                               // Now build the request data
                               #V_PN_Measurement_Data_2.Service_Data_Request.Count_Meas_Values := INT_TO_BYTE(#RECORD_PE_COUNT_MEAS_2);
                               #V_PN_Measurement_Data_2.Service_Data_Request.Meas_Values[PE_ID_F_MAX] := 61;
                               #V_PN_Measurement_Data_2.Service_Data_Request.Meas_Values[PE_ID_U_AVG_L_N_MAX] := 62;
                               #V_PN_Measurement_Data_2.Service_Data_Request.Meas_Values[PE_ID_U_AVG_L_L_MAX] := 63;
                               #V_PN_Measurement_Data_2.Service_Data_Request.Meas_Values[PE_ID_I_AVG_MAX] := 64;
                               #V_PN_Measurement_Data_2.Service_Data_Request.Meas_Values[PE_ID_P_OVERALL_MAX] := 65;
                               #V_PN_Measurement_Data_2.Service_Data_Request.Meas_Values[PE_ID_Q_OVERALL_MAX] := 66;
                               #V_PN_Measurement_Data_2.Service_Data_Request.Meas_Values[PE_ID_S_OVERALL_MAX] := 67;
                               #V_PN_Measurement_Data_2.Service_Data_Request.Meas_Values[PE_ID_COS_OVERALL_MAX] := 68;

                               // Get the minimum values
                               #V_PN_Measurement_Data_2.Service_Data_Request.Meas_Values[PE_ID_U_L1_MIN] := 70;
                               #V_PN_Measurement_Data_2.Service_Data_Request.Meas_Values[PE_ID_U_L2_MIN] := 71;
                               #V_PN_Measurement_Data_2.Service_Data_Request.Meas_Values[PE_ID_U_L3_MIN] := 72;
                               #V_PN_Measurement_Data_2.Service_Data_Request.Meas_Values[PE_ID_U_L1_L2_MIN] := 73;
                               #V_PN_Measurement_Data_2.Service_Data_Request.Meas_Values[PE_ID_U_L2_L3_MIN] := 74;
                               #V_PN_Measurement_Data_2.Service_Data_Request.Meas_Values[PE_ID_U_L3_L1_MIN] := 75;
                               #V_PN_Measurement_Data_2.Service_Data_Request.Meas_Values[PE_ID_I_L1_MIN] := 76;
                               #V_PN_Measurement_Data_2.Service_Data_Request.Meas_Values[PE_ID_I_L2_MIN] := 77;
                               #V_PN_Measurement_Data_2.Service_Data_Request.Meas_Values[PE_ID_I_L3_MIN] := 78;
                               #V_PN_Measurement_Data_2.Service_Data_Request.Meas_Values[PE_ID_S_L1_MIN] := 79;
                               #V_PN_Measurement_Data_2.Service_Data_Request.Meas_Values[PE_ID_S_L2_MIN] := 80;
                               #V_PN_Measurement_Data_2.Service_Data_Request.Meas_Values[PE_ID_S_L3_MIN] := 81;
                               #V_PN_Measurement_Data_2.Service_Data_Request.Meas_Values[PE_ID_P_L1_MIN] := 82;
                               #V_PN_Measurement_Data_2.Service_Data_Request.Meas_Values[PE_ID_P_L2_MIN] := 83;
                               #V_PN_Measurement_Data_2.Service_Data_Request.Meas_Values[PE_ID_P_L3_MIN] := 84;
                               #V_PN_Measurement_Data_2.Service_Data_Request.Meas_Values[PE_ID_Q_L1_MIN] := 85;
                               #V_PN_Measurement_Data_2.Service_Data_Request.Meas_Values[PE_ID_Q_L2_MIN] := 86;
                               #V_PN_Measurement_Data_2.Service_Data_Request.Meas_Values[PE_ID_Q_L3_MIN] := 87;
                               #V_PN_Measurement_Data_2.Service_Data_Request.Meas_Values[PE_ID_COS_L1_MIN] := 88;
                               #V_PN_Measurement_Data_2.Service_Data_Request.Meas_Values[PE_ID_COS_L2_MIN] := 89;
                               #V_PN_Measurement_Data_2.Service_Data_Request.Meas_Values[PE_ID_COS_L3_MIN] := 90;
                               #V_PN_Measurement_Data_2.Service_Data_Request.Meas_Values[PE_ID_F_MIN] := 91;
                               #V_PN_Measurement_Data_2.Service_Data_Request.Meas_Values[PE_ID_U_AVG_L_N_MIN] := 92;
                               #V_PN_Measurement_Data_2.Service_Data_Request.Meas_Values[PE_ID_U_AVG_L_L_MIN] := 93;
                               #V_PN_Measurement_Data_2.Service_Data_Request.Meas_Values[PE_ID_I_AVG_MIN] := 94;
                               #V_PN_Measurement_Data_2.Service_Data_Request.Meas_Values[PE_ID_P_OVERALL_MIN] := 95;
                               #V_PN_Measurement_Data_2.Service_Data_Request.Meas_Values[PE_ID_Q_OVERALL_MIN] := 96;
                               #V_PN_Measurement_Data_2.Service_Data_Request.Meas_Values[PE_ID_S_OVERALL_MIN] := 97;
                               #V_PN_Measurement_Data_2.Service_Data_Request.Meas_Values[PE_ID_COS_OVERALL_MIN] := 98;

                               // Get the energy counter
                               #V_PN_Measurement_Data_2.Service_Data_Request.Meas_Values[PE_ID_E_P_IMP_64] := 210;
                               #V_PN_Measurement_Data_2.Service_Data_Request.Meas_Values[PE_ID_E_P_EXP_64] := 211;
                               #V_PN_Measurement_Data_2.Service_Data_Request.Meas_Values[PE_ID_E_Q_IMP_64] := 212;
                               #V_PN_Measurement_Data_2.Service_Data_Request.Meas_Values[PE_ID_E_Q_EXP_64] := 213;
                               #V_PN_Measurement_Data_2.Service_Data_Request.Meas_Values[PE_ID_E_S_IMP_64] := 214;

                               // Configure the data record number and the length of the data record
                               #Wr_Rec_Index := WORD_TO_INT(#RECORD_PROFIENERGY_INDEX);
                               #Wr_Rec_Max_Length := #RECORD_PE_WRITE_LEN_2;
                               #V_PN_Measurement_Data_2.Block_Header.Block_Length := #RECORD_PE_WRITE_LEN_2 - 4;

                               // Start the writing of the configuration data
                               #Write_Data_Rec_Request := TRUE;

                               // Go to the state for waiting for the answer
                               #Sm_State_Next := #SM_WRITE_MEAS_PN_WAIT_RESP;
                           END_IF;

                           // The PAC is connected with 2
                       ELSIF (#Comm_Type = #PROFIBUS) THEN

                           // The default value for a not measured value is DW16FFFF_FFFF
                           // ==> replace it with 0.0
                           // ==> Therefore check every value in a FOR-loop if it is the default value
                           FOR #Index := 1 TO 47 BY 1 DO
                               IF (#V_DP_Meas_Reset.Meas_Values[#Index] = DW#16#FFFF_FFFF) THEN
                                   #V_DP_Meas_Reset.Meas_Values[#Index] := DW#16#0;
                               ELSE
                                   ; // Value is correct
                               END_IF;
                           END_FOR;

                           // Copy the data to the output structure of the measurement values
                           // but only a view variables can be updated, cause only few of them
                           // are supported by the Energy Meter

                           // ================================================
                           // Proceed the voltage values for each phase
                           // ================================================
                           #Driver_Data.U_L1 := #V_DP_Meas_Data_Res.U_L1;
                           #Driver_Data.U_L2 := #V_DP_Meas_Data_Res.U_L2;
                           #Driver_Data.U_L3 := #V_DP_Meas_Data_Res.U_L3;
                           #Driver_Data.U_PH_N_Average := #V_DP_Meas_Data_Res.U_PH_N_Average;

                           // ================================================
                           // Proceed the voltage values for phase to phase
                           // ================================================
                           #Driver_Data.U_L1_L2 := #V_DP_Meas_Data_Res.U_L1_L2;
                           #Driver_Data.U_L2_L3 := #V_DP_Meas_Data_Res.U_L2_L3;
                           #Driver_Data.U_L3_L1 := #V_DP_Meas_Data_Res.U_L3_L1;
                           #Driver_Data.U_PH_PH_Average := #V_DP_Meas_Data_Res.U_PH_PH_Average;

                           // ================================================
                           // Proceed the current for each phase
                           // ================================================
                           #Driver_Data.I_L1 := #V_DP_Meas_Data_Res.I_L1;
                           #Driver_Data.I_L2 := #V_DP_Meas_Data_Res.I_L2;
                           #Driver_Data.I_L3 := #V_DP_Meas_Data_Res.I_L3;
                           #Driver_Data.I_Average := #V_DP_Meas_Data_Res.I_Average;

                           // ================================================
                           // Proceed the frequency for the complete net
                           // ================================================
                           #Driver_Data.f := #V_DP_Meas_Data_Res.f;

                           // ================================================
                           // Proceed the cos for each phase
                           // ================================================
                           #Driver_Data.Cos_L1 := #V_DP_Meas_Data_Res.Cos_L1;
                           #Driver_Data.Cos_L2 := #V_DP_Meas_Data_Res.Cos_L2;
                           #Driver_Data.Cos_L3 := #V_DP_Meas_Data_Res.Cos_L3;
                           #Driver_Data.Cos_Total := #V_DP_Meas_Data_Res.Cos_Total;

                           // ================================================
                           // Proceed the apparent power for each phase
                           // ================================================
                           #Driver_Data.S_L1 := #V_DP_Meas_Data_Res.S_L1;
                           #Driver_Data.S_L2 := #V_DP_Meas_Data_Res.S_L2;
                           #Driver_Data.S_L3 := #V_DP_Meas_Data_Res.S_L3;
                           #Driver_Data.S_Total := #V_DP_Meas_Data_Res.S_Total;

                           // ================================================
                           // Proceed the reactive power for each phase
                           // ================================================
                           #Driver_Data.Q_L1 := #V_DP_Meas_Data_Res.Q_L1;
                           #Driver_Data.Q_L2 := #V_DP_Meas_Data_Res.Q_L2;
                           #Driver_Data.Q_L3 := #V_DP_Meas_Data_Res.Q_L3;
                           #Driver_Data.Q_Total := #V_DP_Meas_Data_Res.Q_Total;

                           // ================================================
                           // Proceed the effective power for each phase
                           // ================================================
                           #Driver_Data.P_L1 := #V_DP_Meas_Data_Res.P_L1;
                           #Driver_Data.P_L2 := #V_DP_Meas_Data_Res.P_L2;
                           #Driver_Data.P_L3 := #V_DP_Meas_Data_Res.P_L3;
                           #Driver_Data.P_Total := #V_DP_Meas_Data_Res.P_Total;

                           // ================================================
                           // Proceed the energy counter overall
                           // ================================================
                           // Convert the LREAL values to REAL values
                           #LREAL_TO_DINT(id_hdword := #V_DP_Meas_Data_Res.E_Active_Rate1_Im_HW
                                         , id_ldword := #V_DP_Meas_Data_Res.E_Active_Rate1_Im_LW
                           );
                           #Driver_Data.E_Active_Rate1_Import := DINT_TO_REAL(#LREAL_TO_DINT.FINE);
                           #Energy_Counter.Active_Rate1_Imp_Fine := #LREAL_TO_DINT.FINE;
                           #Energy_Counter.Active_Rate1_Imp_Raw := #LREAL_TO_DINT.RAW;

                           #LREAL_TO_DINT(id_hdword := #V_DP_Meas_Data_Res.E_Active_Rate1_Ex_HW
                                         , id_ldword := #V_DP_Meas_Data_Res.E_Active_Rate1_Ex_LW
                           );
                           #Driver_Data.E_Active_Rate1_Export := DINT_TO_REAL(#LREAL_TO_DINT.FINE);
                           #Energy_Counter.Active_Rate1_Exp_Fine := #LREAL_TO_DINT.FINE;
                           #Energy_Counter.Active_Rate1_Exp_Raw := #LREAL_TO_DINT.RAW;

                           #LREAL_TO_DINT(id_hdword := #V_DP_Meas_Data_Res.E_Active_Rate2_Im_HW
                                         , id_ldword := #V_DP_Meas_Data_Res.E_Active_Rate2_Im_LW
                           );
                           #Driver_Data.E_Active_Rate2_Import := DINT_TO_REAL(#LREAL_TO_DINT.FINE);
                           #Energy_Counter.Active_Rate2_Imp_Fine := #LREAL_TO_DINT.FINE;
                           #Energy_Counter.Active_Rate2_Imp_Raw := #LREAL_TO_DINT.RAW;

                           #LREAL_TO_DINT(id_hdword := #V_DP_Meas_Data_Res.E_Active_Rate2_Ex_HW
                                         , id_ldword := #V_DP_Meas_Data_Res.E_Active_Rate2_Ex_LW
                           );
                           #Driver_Data.E_Active_Rate2_Export := DINT_TO_REAL(#LREAL_TO_DINT.FINE);
                           #Energy_Counter.Active_Rate2_Exp_Fine := #LREAL_TO_DINT.FINE;
                           #Energy_Counter.Active_Rate2_Exp_Raw := #LREAL_TO_DINT.RAW;

                           #LREAL_TO_DINT(id_hdword := #V_DP_Meas_Data_Res.E_Reactive_Rate1_Im_HW
                                         , id_ldword := #V_DP_Meas_Data_Res.E_Reactive_Rate1_Im_LW
                           );
                           #Driver_Data.E_Reactive_Rate1_Import := DINT_TO_REAL(#LREAL_TO_DINT.FINE);
                           #Energy_Counter.Reactive_Rate1_Imp_Fine := #LREAL_TO_DINT.FINE;
                           #Energy_Counter.Reactive_Rate1_Imp_Raw := #LREAL_TO_DINT.RAW;

                           #LREAL_TO_DINT(id_hdword := #V_DP_Meas_Data_Res.E_Reactive_Rate1_Ex_HW
                                         , id_ldword := #V_DP_Meas_Data_Res.E_Reactive_Rate1_Ex_LW
                           );
                           #Driver_Data.E_Reactive_Rate1_Export := DINT_TO_REAL(#LREAL_TO_DINT.FINE);
                           #Energy_Counter.Reactive_Rate1_Exp_Fine := #LREAL_TO_DINT.FINE;
                           #Energy_Counter.Reactive_Rate1_Exp_Raw := #LREAL_TO_DINT.RAW;

                           #LREAL_TO_DINT(id_hdword := #V_DP_Meas_Data_Res.E_Reactive_Rate2_Im_HW
                                         , id_ldword := #V_DP_Meas_Data_Res.E_Reactive_Rate2_Im_LW
                           );
                           #Driver_Data.E_Reactive_Rate2_Import := DINT_TO_REAL(#LREAL_TO_DINT.FINE);
                           #Energy_Counter.Reactive_Rate2_Imp_Fine := #LREAL_TO_DINT.FINE;
                           #Energy_Counter.Reactive_Rate2_Imp_Raw := #LREAL_TO_DINT.RAW;

                           #LREAL_TO_DINT(id_hdword := #V_DP_Meas_Data_Res.E_Reactive_Rate2_Ex_HW
                                         , id_ldword := #V_DP_Meas_Data_Res.E_Reactive_Rate2_Ex_LW
                           );
                           #Driver_Data.E_Reactive_Rate2_Export := DINT_TO_REAL(#LREAL_TO_DINT.FINE);
                           #Energy_Counter.Reactive_Rate2_Exp_Fine := #LREAL_TO_DINT.FINE;
                           #Energy_Counter.Reactive_Rate2_Exp_Raw := #LREAL_TO_DINT.RAW;

                           #LREAL_TO_DINT(id_hdword := #V_DP_Meas_Data_Res.E_Apparent_Rate1_Im_HW
                                         , id_ldword := #V_DP_Meas_Data_Res.E_Apparent_Rate1_Im_LW
                           );
                           #Driver_Data.E_Apparent_Rate1_Import := DINT_TO_REAL(#LREAL_TO_DINT.FINE);
                           #Energy_Counter.Apparent_Rate1_Imp_Fine := #LREAL_TO_DINT.FINE;
                           #Energy_Counter.Apparent_Rate1_Imp_Raw := #LREAL_TO_DINT.RAW;

                           #LREAL_TO_DINT(id_hdword := #V_DP_Meas_Data_Res.E_Apparent_Rate2_Im_HW
                                         , id_ldword := #V_DP_Meas_Data_Res.E_Apparent_Rate2_Im_LW
                           );
                           #Driver_Data.E_Apparent_Rate2_Import := DINT_TO_REAL(#LREAL_TO_DINT.FINE);
                           #Energy_Counter.Apparent_Rate2_Imp_Fine := #LREAL_TO_DINT.FINE;
                           #Energy_Counter.Apparent_Rate2_Imp_Raw := #LREAL_TO_DINT.RAW;

                           // The minimum and maximum values should be calculated in the driver
                           IF (#Min_Max_Calculated = TRUE) THEN

                               // Save the time to update the values
                               #Time_to_update := #Time_Measurement.ET;

                               // Reset the timer to restart the time next time
                               #Time_Measurement(IN := FALSE,
                                                 PT := T#21d);

                               // Read the current time to set the timestamp of the measurement values
                               #General_Ret_Val := RD_SYS_T(OUT => #Time_Stamp_Meas_Values);

                               // Release the communication resource
                               #Comm_Resource_Counter := #Comm_Resource_Counter - 1;

                               //===========================================================================
                               //====== Generate the minimum and maximum values ============================
                               //===========================================================================

                               // ================================================
                               // Proceed the voltage values for each phase
                               // ================================================

                               // Check the voltage values for the phases for a new maximum or minimum
                               // Phase L1
                               IF (#Driver_Data.U_L1 > #Driver_Data.U_L1_max) THEN
                                   #Driver_Data.U_L1_max := #Driver_Data.U_L1;
                               ELSIF (#Driver_Data.U_L1 < #Driver_Data.U_L1_min) THEN
                                   #Driver_Data.U_L1_min := #Driver_Data.U_L1;
                               ELSE
                                   ; // No new maximum or minimum value
                               END_IF;

                               // Phase L2
                               IF (#Driver_Data.U_L2 > #Driver_Data.U_L2_max) THEN
                                   #Driver_Data.U_L2_max := #Driver_Data.U_L2;
                               ELSIF (#Driver_Data.U_L2 < #Driver_Data.U_L2_min) THEN
                                   #Driver_Data.U_L2_min := #Driver_Data.U_L2;
                               ELSE
                                   ; // No new maximum or minimum value
                               END_IF;

                               // Phase L3
                               IF (#Driver_Data.U_L3 > #Driver_Data.U_L3_max) THEN
                                   #Driver_Data.U_L3_max := #Driver_Data.U_L3;
                               ELSIF (#Driver_Data.U_L3 < #Driver_Data.U_L3_min) THEN
                                   #Driver_Data.U_L3_min := #Driver_Data.U_L3;
                               ELSE
                                   ; // No new maximum or minimum value
                               END_IF;

                               // Check the voltage average value of the phases for a new maximum or minimum
                               // Average value
                               IF (#Driver_Data.U_PH_N_Average > #Driver_Data.U_PH_N_Average_max) THEN
                                   #Driver_Data.U_PH_N_Average_max := #Driver_Data.U_PH_N_Average;
                               ELSIF (#Driver_Data.U_PH_N_Average < #Driver_Data.U_PH_N_Average_min) THEN
                                   #Driver_Data.U_PH_N_Average_min := #Driver_Data.U_PH_N_Average;
                               ELSE
                                   ; // No new maximum or minimum value
                               END_IF;

                               // ================================================
                               // Proceed the voltage values for phase to phase
                               // ================================================

                               // Check the voltage values for the phases for a new maximum or minimum
                               // Phase L1 - L2
                               IF (#Driver_Data.U_L1_L2 > #Driver_Data.U_L1_L2_max) THEN
                                   #Driver_Data.U_L1_L2_max := #Driver_Data.U_L1_L2;
                               ELSIF (#Driver_Data.U_L1_L2 < #Driver_Data.U_L1_L2_min) THEN
                                   #Driver_Data.U_L1_L2_min := #Driver_Data.U_L1_L2;
                               ELSE
                                   ; // No new maximum or minimum value
                               END_IF;

                               // Phase L2 - L3
                               IF (#Driver_Data.U_L2_L3 > #Driver_Data.U_L2_L3_max) THEN
                                   #Driver_Data.U_L2_L3_max := #Driver_Data.U_L2_L3;
                               ELSIF (#Driver_Data.U_L2_L3 < #Driver_Data.U_L2_L3_min) THEN
                                   #Driver_Data.U_L2_L3_min := #Driver_Data.U_L2_L3;
                               ELSE
                                   ; // No new maximum or minimum value
                               END_IF;

                               // Phase L3 - L1
                               IF (#Driver_Data.U_L3_L1 > #Driver_Data.U_L3_L1_max) THEN
                                   #Driver_Data.U_L3_L1_max := #Driver_Data.U_L3_L1;
                               ELSIF (#Driver_Data.U_L3_L1 < #Driver_Data.U_L3_L1_min) THEN
                                   #Driver_Data.U_L3_L1_min := #Driver_Data.U_L3_L1;
                               ELSE
                                   ; // No new maximum or minimum value
                               END_IF;

                               // Check the voltage average value of the phases for a new maximum or minimum
                               // Average value
                               IF (#Driver_Data.U_PH_PH_Average > #Driver_Data.U_PH_PH_Average_max) THEN
                                   #Driver_Data.U_PH_PH_Average_max := #Driver_Data.U_PH_PH_Average;
                               ELSIF (#Driver_Data.U_PH_PH_Average < #Driver_Data.U_PH_PH_Average_min) THEN
                                   #Driver_Data.U_PH_PH_Average_min := #Driver_Data.U_PH_PH_Average;
                               ELSE
                                   ; // No new maximum or minimum value
                               END_IF;

                               // ================================================
                               // Proceed the current for each phase
                               // ================================================

                               // Check the current values for the phases for a new maximum or minimum
                               // Phase L1
                               IF (#Driver_Data.I_L1 > #Driver_Data.I_L1_max) THEN
                                   #Driver_Data.I_L1_max := #Driver_Data.I_L1;
                               ELSIF (#Driver_Data.I_L1 < #Driver_Data.I_L1_min) THEN
                                   #Driver_Data.I_L1_min := #Driver_Data.I_L1;
                               ELSE
                                   ; // No new maximum or minimum value
                               END_IF;

                               // Phase L2
                               IF (#Driver_Data.I_L2 > #Driver_Data.I_L2_max) THEN
                                   #Driver_Data.I_L2_max := #Driver_Data.I_L2;
                               ELSIF (#Driver_Data.I_L2 < #Driver_Data.I_L2_min) THEN
                                   #Driver_Data.I_L2_min := #Driver_Data.I_L2;
                               ELSE
                                   ; // No new maximum or minimum value
                               END_IF;

                               // Phase L3
                               IF (#Driver_Data.I_L3 > #Driver_Data.I_L3_max) THEN
                                   #Driver_Data.I_L3_max := #Driver_Data.I_L3;
                               ELSIF (#Driver_Data.I_L3 < #Driver_Data.I_L3_min) THEN
                                   #Driver_Data.I_L3_min := #Driver_Data.I_L3;
                               ELSE
                                   ; // No new maximum or minimum value
                               END_IF;

                               // Check the voltage average value of the phases for a new maximum or minimum
                               // Average value
                               IF (#Driver_Data.I_Average > #Driver_Data.I_Average_max) THEN
                                   #Driver_Data.I_Average_max := #Driver_Data.I_Average;
                               ELSIF (#Driver_Data.I_Average < #Driver_Data.I_Average_min) THEN
                                   #Driver_Data.I_Average_min := #Driver_Data.I_Average;
                               ELSE
                                   ; // No new maximum or minimum value
                               END_IF;

                               // ================================================
                               // Proceed the frequency for the complete net
                               // ================================================

                               // Check the frequency values for the phases for a new maximum or minimum
                               IF (#Driver_Data.f > #Driver_Data.f_max) THEN
                                   #Driver_Data.f_max := #Driver_Data.f;
                               ELSIF (#Driver_Data.f < #Driver_Data.f_min) THEN
                                   #Driver_Data.f_min := #Driver_Data.f;
                               ELSE
                                   ; // No new maximum or minimum value
                               END_IF;

                               // ================================================
                               // Proceed the cos for each phase
                               // ================================================

                               // Check the power factor values for the phases for a new maximum or minimum
                               // Phase L1
                               IF (#Driver_Data.Cos_L1 > #Driver_Data.Cos_L1_max) THEN
                                   #Driver_Data.Cos_L1_max := #Driver_Data.Cos_L1;
                               ELSIF (#Driver_Data.Cos_L1 < #Driver_Data.Cos_L1_min) THEN
                                   #Driver_Data.Cos_L1_min := #Driver_Data.Cos_L1;
                               ELSE
                                   ; // No new maximum or minimum value
                               END_IF;

                               // Phase L2
                               IF (#Driver_Data.Cos_L2 > #Driver_Data.Cos_L2_max) THEN
                                   #Driver_Data.Cos_L2_max := #Driver_Data.Cos_L2;
                               ELSIF (#Driver_Data.Cos_L2 < #Driver_Data.Cos_L2_min) THEN
                                   #Driver_Data.Cos_L2_min := #Driver_Data.Cos_L2;
                               ELSE
                                   ; // No new maximum or minimum value
                               END_IF;

                               // Phase L3
                               IF (#Driver_Data.Cos_L3 > #Driver_Data.Cos_L3_max) THEN
                                   #Driver_Data.Cos_L3_max := #Driver_Data.Cos_L3;
                               ELSIF (#Driver_Data.Cos_L3 < #Driver_Data.Cos_L3_min) THEN
                                   #Driver_Data.Cos_L3_min := #Driver_Data.Cos_L3;
                               ELSE
                                   ; // No new maximum or minimum value
                               END_IF;

                               // Overall
                               IF (#Driver_Data.Cos_Total > #Driver_Data.Cos_Total_max) THEN
                                   #Driver_Data.Cos_Total_max := #Driver_Data.Cos_Total;
                               ELSIF (#Driver_Data.Cos_Total < #Driver_Data.Cos_Total_min) THEN
                                   #Driver_Data.Cos_Total_min := #Driver_Data.Cos_Total;
                               ELSE
                                   ; // No new maximum or minimum value
                               END_IF;

                               // ================================================
                               // Proceed the apparent power for each phase
                               // ================================================

                               // Check the apparent power values for the phases for a new maximum or minimum
                               // Phase L1
                               IF (#Driver_Data.S_L1 > #Driver_Data.S_L1_max) THEN
                                   #Driver_Data.S_L1_max := #Driver_Data.S_L1;
                               ELSIF (#Driver_Data.S_L1 < #Driver_Data.S_L1_min) THEN
                                   #Driver_Data.S_L1_min := #Driver_Data.S_L1;
                               ELSE
                                   ; // No new maximum or minimum value
                               END_IF;

                               // Phase L2
                               IF (#Driver_Data.S_L2 > #Driver_Data.S_L2_max) THEN
                                   #Driver_Data.S_L2_max := #Driver_Data.S_L2;
                               ELSIF (#Driver_Data.S_L2 < #Driver_Data.S_L2_min) THEN
                                   #Driver_Data.S_L2_min := #Driver_Data.S_L2;
                               ELSE
                                   ; // No new maximum or minimum value
                               END_IF;

                               // Phase L3
                               IF (#Driver_Data.S_L3 > #Driver_Data.S_L3_max) THEN
                                   #Driver_Data.S_L3_max := #Driver_Data.S_L3;
                               ELSIF (#Driver_Data.S_L3 < #Driver_Data.S_L3_min) THEN
                                   #Driver_Data.S_L3_min := #Driver_Data.S_L3;
                               ELSE
                                   ; // No new maximum or minimum value
                               END_IF;

                               // Overall
                               IF (#Driver_Data.S_Total > #Driver_Data.S_Total_max) THEN
                                   #Driver_Data.S_Total_max := #Driver_Data.S_Total;
                               ELSIF (#Driver_Data.S_Total < #Driver_Data.S_Total_min) THEN
                                   #Driver_Data.S_Total_min := #Driver_Data.S_Total;
                               ELSE
                                   ; // No new maximum or minimum value
                               END_IF;

                               // ================================================
                               // Proceed the reactive power for each phase
                               // ================================================

                               // Check the reactive power values for the phases for a new maximum or minimum
                               // Phase L1
                               IF (#Driver_Data.Q_L1 > #Driver_Data.Q_L1_max) THEN
                                   #Driver_Data.Q_L1_max := #Driver_Data.Q_L1;
                               ELSIF (#Driver_Data.Q_L1 < #Driver_Data.Q_L1_min) THEN
                                   #Driver_Data.Q_L1_min := #Driver_Data.Q_L1;
                               ELSE
                                   ; // No new maximum or minimum value
                               END_IF;

                               // Phase L2
                               IF (#Driver_Data.Q_L2 > #Driver_Data.Q_L2_max) THEN
                                   #Driver_Data.Q_L2_max := #Driver_Data.Q_L2;
                               ELSIF (#Driver_Data.Q_L2 < #Driver_Data.Q_L2_min) THEN
                                   #Driver_Data.Q_L2_min := #Driver_Data.Q_L2;
                               ELSE
                                   ; // No new maximum or minimum value
                               END_IF;

                               // Phase L3
                               IF (#Driver_Data.Q_L3 > #Driver_Data.Q_L3_max) THEN
                                   #Driver_Data.Q_L3_max := #Driver_Data.Q_L3;
                               ELSIF (#Driver_Data.Q_L3 < #Driver_Data.Q_L3_min) THEN
                                   #Driver_Data.Q_L3_min := #Driver_Data.Q_L3;
                               ELSE
                                   ; // No new maximum or minimum value
                               END_IF;

                               // Overall
                               IF (#Driver_Data.Q_Total > #Driver_Data.Q_Total_max) THEN
                                   #Driver_Data.Q_Total_max := #Driver_Data.Q_Total;
                               ELSIF (#Driver_Data.Q_Total < #Driver_Data.Q_Total_min) THEN
                                   #Driver_Data.Q_Total_min := #Driver_Data.Q_Total;
                               ELSE
                                   ; // No new maximum or minimum value
                               END_IF;

                               // ================================================
                               // Proceed the effective power for each phase
                               // ================================================

                               // Check the effective power values for the phases for a new maximum or minimum
                               // Phase L1
                               IF (#Driver_Data.P_L1 > #Driver_Data.P_L1_max) THEN
                                   #Driver_Data.P_L1_max := #Driver_Data.P_L1;
                               ELSIF (#Driver_Data.P_L1 < #Driver_Data.P_L1_min) THEN
                                   #Driver_Data.P_L1_min := #Driver_Data.P_L1;
                               ELSE
                                   ; // No new maximum or minimum value
                               END_IF;

                               // Phase L2
                               IF (#Driver_Data.P_L2 > #Driver_Data.P_L2_max) THEN
                                   #Driver_Data.P_L2_max := #Driver_Data.P_L2;
                               ELSIF (#Driver_Data.P_L2 < #Driver_Data.P_L2_min) THEN
                                   #Driver_Data.P_L2_min := #Driver_Data.P_L2;
                               ELSE
                                   ; // No new maximum or minimum value
                               END_IF;

                               // Phase L3
                               IF (#Driver_Data.P_L3 > #Driver_Data.P_L3_max) THEN
                                   #Driver_Data.P_L3_max := #Driver_Data.P_L3;
                               ELSIF (#Driver_Data.P_L3 < #Driver_Data.P_L3_min) THEN
                                   #Driver_Data.P_L3_min := #Driver_Data.P_L3;
                               ELSE
                                   ; // No new maximum or minimum value
                               END_IF;

                               // Overall
                               IF (#Driver_Data.P_Total > #Driver_Data.P_Total_max) THEN
                                   #Driver_Data.P_Total_max := #Driver_Data.P_Total;
                               ELSIF (#Driver_Data.P_Total < #Driver_Data.P_Total_min) THEN
                                   #Driver_Data.P_Total_min := #Driver_Data.P_Total;
                               ELSE
                                   ; // No new maximum or minimum value
                               END_IF;

                               // Go back to the main state and wait for a new request
                               #Sm_State_Next := #SM_IDLE;
                           ELSE

                               // In the second reading, get the min max values from the SENTRON PAC.
                               // ==> Configure the data record, to get the values by using the block reading of more values with one command

                               // In the first block, read the max values for voltage, current, apparent power, effective power, reactive power and the power factor
                               // The ID of the first measurement value to read is 75.
                               // 21 values will be read, length = 21*4 = 84 / 2 (unit is amount of words) = 42
                               #V_DP_Measurement_Data.Measurement_Data[1].Measurement_ID := 75;
                               #V_DP_Measurement_Data.Measurement_Data[1].Measurement_Len := 42;

                               // In the second block, read the max values for net frequency, the average values and the overall power values
                               // and all minimum values
                               // The ID of the first measurement value to read is 129.
                               // 8 values will be read, length = 37*4 = 148 / 2 (unit is amount of words) = 74
                               #V_DP_Measurement_Data.Measurement_Data[2].Measurement_ID := 129;
                               #V_DP_Measurement_Data.Measurement_Data[2].Measurement_Len := 74;

                               // Configure the data record number and the length of the data record
                               #Wr_Rec_Index := #RECORD_47_FLEX_ACCESS_MEASUREMENT_INDEX;
                               #Wr_Rec_Max_Length := #RECORD_47_WRITE_MINMAX_LEN;

                               // Start the writing of the configuration data
                               #Write_Data_Rec_Request := TRUE;

                               // Go to the state for waiting for the answer
                               #Sm_State_Next := #SM_WRITE_MINMAX_WAIT_RESP;
                           END_IF;
                       ELSE
                           ; // Further communication methods
                       END_IF;
                   ELSE
                       ; // Reading still in progress
                   END_IF;

                   // Wait for the answer of the SENTRON PAC
               #SM_WRITE_MEAS_PN_WAIT_RESP:

                   // Set the state of the block to "Reading the measurement values"
                   #Error_Location := #STATUS_READ_MEAS;

                   // Start the watchdog, while waiting for a response
                   #Watchdog_Run := TRUE;

                   // The configuration of the data record 47 on the PAC 4200 failed with an error
                   IF ((#Write_Data_Record.ERROR = TRUE)
                       OR (#Watchdog.Q = TRUE)) THEN

                       // Reset the watchdog
                       #Watchdog_Run := FALSE;

                       // Save the error code for the user to display the error reason and location
                       #Error_Location := #ERR_LOC_WRITE_MEAS_2;
                       #Error_Code := #Write_Data_Record.STATUS;

                       // Reset the request bit to write a record to the Energy Meter for
                       // generating a positive edge with the next request
                       #Write_Data_Rec_Request := FALSE;

                       // Release the communication resource
                       #Comm_Resource_Counter := #Comm_Resource_Counter - 1;

                       // Go back to the main state and wait for a new request
                       #Sm_State_Next := #SM_IDLE;

                       // The configuration of the data record 47 on the PAC 4200 has been finished with success
                   ELSIF (#Write_Data_Record.DONE = TRUE) THEN

                       // Reset the watchdog
                       #Watchdog_Run := FALSE;

                       // Reset the error code and location
                       #Error_Code := DW#16#0000_0000;

                       // Reset the request bit to write a record to the SENTRON PAC 4200 for
                       // generating a positive edge with the next request
                       #Write_Data_Rec_Request := FALSE;

                       // Now configure the values to read these measurement values
                       #Rd_Rec_Index := WORD_TO_INT(#RECORD_PROFIENERGY_INDEX);
                       #Rd_Rec_Max_Length := #RECORD_PE_READ_LEN_2;

                       // Start the reading of the measurement values
                       #Read_Data_Rec_Request := TRUE;

                       // Go back to the main state and wait for a new request
                       #Sm_State_Next := #SM_READ_MEAS_PN_WAIT_RESP;
                   ELSE
                       ; // Reading still in progress
                   END_IF;

                   // The wait state after an error
               #SM_READ_MEAS_PN_WAIT_TIME:

                   // The timer has to run
                   #Error_Retry_Timer_Run := TRUE;

                   // If the timer elapsed, retry reading
                   IF (#Error_Retry_Timer.Q = TRUE) THEN

                       // Retry the reading
                       #Sm_State_Next := #SM_READ_MEAS_PN_WAIT_RESP;
                   ELSE
                       ; // Still wait
                   END_IF;

                   // Wait for an answer of the reading of the current measuement values
               #SM_READ_MEAS_PN_WAIT_RESP:

                   // Start the watchdog, while waiting for a response
                   #Watchdog_Run := TRUE;

                   // Set the request to true, if the bit is reset in case of an error
                   #Read_Data_Rec_Request := #Error_Retry_Timer.Q;

                   // The update of the data failed with an error
                   IF ((#Read_Data_Record.ERROR = TRUE)
                       OR (#Watchdog.Q = TRUE)) THEN

                       // Reset the request bit to read a record from the Energy Meter for
                       // generating a positive edge with the next request
                       #Read_Data_Rec_Request := FALSE;

                       // Increase the retries to get an answer
                       #Error_Retry_Counter := #Error_Retry_Counter + 1;

                       // Check if the device is still busy
                       IF (((#Read_Data_Record.STATUS = #ERROR_CODE_DEVICE_BUSY)
                           AND (#Error_Retry_Counter >= #ERROR_RETRY_LIMIT))
                           OR (#Read_Data_Record.STATUS <> #ERROR_CODE_DEVICE_BUSY)) THEN

                           // Reset the watchdog
                           #Watchdog_Run := FALSE;

                           // Save the time to update the values, even with an error
                           #Time_to_update := #Time_Measurement.ET;

                           // Reset the timer to restart the time next time
                           #Time_Measurement(IN := FALSE,
                                             PT := T#21d);

                           // Reset the timer
                           #Error_Retry_Timer_Run := FALSE;

                           // Reset the retry counter
                           #Error_Retry_Counter := 0;

                           // Save the error code for the user to display the error reason and location
                           #Error_Location := #ERR_LOC_READ_MEAS_2;
                           #Error_Code := #Read_Data_Record.STATUS;

                           // Release the communication resource
                           #Comm_Resource_Counter := #Comm_Resource_Counter - 1;

                           // Go back to the main state and wait for a new request
                           #Sm_State_Next := #SM_IDLE;
                       ELSE
                           // Reset the timer
                           #Error_Retry_Timer(IN := FALSE,
                                              PT := #TIME_RETRY_TIMER);

                           // Start the error timer
                           #Error_Retry_Timer_Run := TRUE;

                           // Go to the wait state
                           #Sm_State_Next := #SM_READ_MEAS_PN_WAIT_TIME;
                       END_IF;

                       // The update of the has been finished with success
                   ELSIF (#Read_Data_Record.VALID = TRUE) THEN

                       // Reset the watchdog
                       #Watchdog_Run := FALSE;

                       // Reset the retry counter
                       #Error_Retry_Counter := 0;

                       // Reset the error code and location
                       #Error_Code := DW#16#0000_0000;

                       // Save the time to update the values
                       #Time_to_update := #Time_Measurement.ET;

                       // Release the communication resource
                       #Comm_Resource_Counter := #Comm_Resource_Counter - 1;

                       // Reset the request bit to read a record from the Energy Meter for
                       // generating a positive edge with the next request
                       #Read_Data_Rec_Request := FALSE;

                       // Check the header of the PROFIenergy response for an error
                       // First of all, check the block type for correctness, it must be W160801
                       IF (#V_PN_Meas_Data_Res_2.Block_Header.Block_Type <> #PN_BLOCK_TYPE_READ) THEN

                           // Set the error code and location
                           #Error_Location := #ERR_LOC_PN_INV_BLOCK_2;
                           #Error_Code := #ERR_CODE_GENERAL;

                           // Check the service request ID ==> it should be 0x10
                       ELSIF (#V_PN_Meas_Data_Res_2.Response_Header.Service_Request_ID <> #PN_REQUEST_ID_GET_MEASUREMENT_VALUES) THEN

                           // Set the error code and location
                           #Error_Location := #ERR_LOC_PN_INVALID_REQUEST_ID_2;
                           #Error_Code := #ERR_CODE_GENERAL;

                           // Check the request reference ==> should be the same as in the request
                       ELSIF (#V_PN_Meas_Data_Res_2.Response_Header.Request_Reference <> #PE_Request_Reference) THEN

                           // Set the error code and location
                           #Error_Location := #ERR_LOC_PN_INV_REQ_REF_2;
                           #Error_Code := #ERR_CODE_GENERAL;

                           // Check the status of the response ==> should be ready (0x01)
                       ELSIF (#V_PN_Meas_Data_Res_2.Service_Header_Response.Status = B#16#02) THEN

                           // Set the error code and location
                           #Error_Location := #ERR_LOC_PN_PE_CMD_FAIL_2;
                           #Error_Code := #Read_Data_Record.STATUS;

                           // Check the data structure identifier ==> should be 0x01
                       ELSIF (#V_PN_Meas_Data_Res_2.Service_Header_Response.Data_Struct_Identifier <> B#16#01) THEN

                           // Set the error code and location
                           #Error_Location := #ERR_LOC_PN_INV_DATSTR_2;
                           #Error_Code := #ERR_CODE_GENERAL;

                           // The header is OK
                       ELSE
                           // Set the state of the block to "Waiting for a new request"
                           #Error_Location := #STATUS_IDLE;

                           // Reset the timer to restart the time next time
                           #Time_Measurement(IN := FALSE,
                                             PT := T#21d);

                           // Read the current time to set the timestamp of the measurement values
                           #General_Ret_Val := RD_SYS_T(OUT => #Time_Stamp_Meas_Values);

                           // The default value for a not measured value is DW16FFFF_FFFF
                           // ==> replace it with 0.0
                           // ==> Therefore check every value in a FOR-loop if it is the default value
                           FOR #Index := 51 TO 87 BY 1 DO
                               IF (REAL_TO_DWORD(#V_PN_Meas_Data_Res_2.Service_Data_Response.Meas_Values_32Bit[#Index].Meas_Value) = DW#16#FFFF_FFFF) THEN
                                   #V_PN_Meas_Data_Res_2.Service_Data_Response.Meas_Values_32Bit[#Index].Meas_Value := 0.0;
                               ELSE
                                   ; // Value is correct
                               END_IF;
                           END_FOR;

                           // Copy the data to the output structure of the measurement values
                           // but only a view variables can be updated, cause only few of them
                           // are supported by the Energy Meter

                           // ================================================
                           // Proceed the energy counter overall
                           // ================================================

                           // Transfer the information to the energy counter structure
                           // Convert the LREAL values to REAL values
                           #LREAL_TO_DINT(id_hdword := #V_PN_Meas_Data_Res_2.Service_Data_Response.Meas_Values_64Bit[PE_ID_E_P_EXP_64].Meas_Value_H,
                                         id_ldword := #V_PN_Meas_Data_Res_2.Service_Data_Response.Meas_Values_64Bit[PE_ID_E_P_EXP_64].Meas_Value_L
                           );
                           #Energy_Counter.Active_Rate1_Exp_Fine := #LREAL_TO_DINT.FINE;
                           #Energy_Counter.Active_Rate1_Exp_Raw := #LREAL_TO_DINT.RAW;
                           #Driver_Data.E_Active_Rate1_Export := DINT_TO_REAL(#LREAL_TO_DINT.FINE);

                           #LREAL_TO_DINT(id_hdword := #V_PN_Meas_Data_Res_2.Service_Data_Response.Meas_Values_64Bit[PE_ID_E_P_IMP_64].Meas_Value_H,
                                         id_ldword := #V_PN_Meas_Data_Res_2.Service_Data_Response.Meas_Values_64Bit[PE_ID_E_P_IMP_64].Meas_Value_L
                           );
                           #Energy_Counter.Active_Rate1_Imp_Fine := #LREAL_TO_DINT.FINE;
                           #Energy_Counter.Active_Rate1_Imp_Raw := #LREAL_TO_DINT.RAW;
                           #Driver_Data.E_Active_Rate1_Import := DINT_TO_REAL(#LREAL_TO_DINT.FINE);

                           #LREAL_TO_DINT(id_hdword := #V_PN_Meas_Data_Res_2.Service_Data_Response.Meas_Values_64Bit[PE_ID_E_Q_EXP_64].Meas_Value_H,
                                         id_ldword := #V_PN_Meas_Data_Res_2.Service_Data_Response.Meas_Values_64Bit[PE_ID_E_Q_EXP_64].Meas_Value_L
                           );
                           #Energy_Counter.Reactive_Rate1_Exp_Fine := #LREAL_TO_DINT.FINE;
                           #Energy_Counter.Reactive_Rate1_Exp_Raw := #LREAL_TO_DINT.RAW;
                           #Driver_Data.E_Reactive_Rate1_Export := DINT_TO_REAL(#LREAL_TO_DINT.FINE);

                           #LREAL_TO_DINT(id_hdword := #V_PN_Meas_Data_Res_2.Service_Data_Response.Meas_Values_64Bit[PE_ID_E_Q_IMP_64].Meas_Value_H,
                                         id_ldword := #V_PN_Meas_Data_Res_2.Service_Data_Response.Meas_Values_64Bit[PE_ID_E_Q_IMP_64].Meas_Value_L
                           );
                           #Energy_Counter.Reactive_Rate1_Imp_Fine := #LREAL_TO_DINT.FINE;
                           #Energy_Counter.Reactive_Rate1_Imp_Raw := #LREAL_TO_DINT.RAW;
                           #Driver_Data.E_Reactive_Rate1_Import := DINT_TO_REAL(#LREAL_TO_DINT.FINE);

                           #LREAL_TO_DINT(id_hdword := #V_PN_Meas_Data_Res_2.Service_Data_Response.Meas_Values_64Bit[PE_ID_E_S_IMP_64].Meas_Value_H,
                                         id_ldword := #V_PN_Meas_Data_Res_2.Service_Data_Response.Meas_Values_64Bit[PE_ID_E_S_IMP_64].Meas_Value_L
                           );
                           #Energy_Counter.Apparent_Rate1_Imp_Fine := #LREAL_TO_DINT.FINE;
                           #Energy_Counter.Apparent_Rate1_Imp_Raw := #LREAL_TO_DINT.RAW;
                           #Driver_Data.E_Apparent_Rate1_Import := DINT_TO_REAL(#LREAL_TO_DINT.FINE);

                           //===========================================================================
                           //====== Generate the minimum and maximum values ============================
                           //===========================================================================

                           // ================================================
                           // Proceed the voltage values for each phase
                           // ================================================
                           #Driver_Data.U_L1_min := #V_PN_Meas_Data_Res_2.Service_Data_Response.Meas_Values_32Bit[PE_ID_U_L1_MIN].Meas_Value;
                           #Driver_Data.U_L2_min := #V_PN_Meas_Data_Res_2.Service_Data_Response.Meas_Values_32Bit[PE_ID_U_L2_MIN].Meas_Value;
                           #Driver_Data.U_L3_min := #V_PN_Meas_Data_Res_2.Service_Data_Response.Meas_Values_32Bit[PE_ID_U_L3_MIN].Meas_Value;
                           #Driver_Data.U_PH_N_Average_max := #V_PN_Meas_Data_Res_2.Service_Data_Response.Meas_Values_32Bit[PE_ID_U_AVG_L_N_MAX].Meas_Value;
                           #Driver_Data.U_PH_N_Average_min := #V_PN_Meas_Data_Res_2.Service_Data_Response.Meas_Values_32Bit[PE_ID_U_AVG_L_N_MIN].Meas_Value;
                           #Driver_Data.U_L1_L2_min := #V_PN_Meas_Data_Res_2.Service_Data_Response.Meas_Values_32Bit[PE_ID_U_L1_L2_MIN].Meas_Value;
                           #Driver_Data.U_L2_L3_min := #V_PN_Meas_Data_Res_2.Service_Data_Response.Meas_Values_32Bit[PE_ID_U_L2_L3_MIN].Meas_Value;
                           #Driver_Data.U_L3_L1_min := #V_PN_Meas_Data_Res_2.Service_Data_Response.Meas_Values_32Bit[PE_ID_U_L3_L1_MIN].Meas_Value;
                           #Driver_Data.U_PH_PH_Average_max := #V_PN_Meas_Data_Res_2.Service_Data_Response.Meas_Values_32Bit[PE_ID_U_AVG_L_L_MAX].Meas_Value;
                           #Driver_Data.U_PH_PH_Average_min := #V_PN_Meas_Data_Res_2.Service_Data_Response.Meas_Values_32Bit[PE_ID_U_AVG_L_L_MIN].Meas_Value;
                           #Driver_Data.I_L1_min := #V_PN_Meas_Data_Res_2.Service_Data_Response.Meas_Values_32Bit[PE_ID_I_L1_MIN].Meas_Value;
                           #Driver_Data.I_L2_min := #V_PN_Meas_Data_Res_2.Service_Data_Response.Meas_Values_32Bit[PE_ID_I_L2_MIN].Meas_Value;
                           #Driver_Data.I_L3_min := #V_PN_Meas_Data_Res_2.Service_Data_Response.Meas_Values_32Bit[PE_ID_I_L3_MIN].Meas_Value;
                           #Driver_Data.I_Average_max := #V_PN_Meas_Data_Res_2.Service_Data_Response.Meas_Values_32Bit[PE_ID_I_AVG_MAX].Meas_Value;
                           #Driver_Data.I_Average_min := #V_PN_Meas_Data_Res_2.Service_Data_Response.Meas_Values_32Bit[PE_ID_I_AVG_MIN].Meas_Value;
                           #Driver_Data.f_max := #V_PN_Meas_Data_Res_2.Service_Data_Response.Meas_Values_32Bit[PE_ID_F_MAX].Meas_Value;
                           #Driver_Data.f_min := #V_PN_Meas_Data_Res_2.Service_Data_Response.Meas_Values_32Bit[PE_ID_F_MIN].Meas_Value;
                           #Driver_Data.Cos_L1_min := #V_PN_Meas_Data_Res_2.Service_Data_Response.Meas_Values_32Bit[PE_ID_COS_L1_MIN].Meas_Value;
                           #Driver_Data.Cos_L2_min := #V_PN_Meas_Data_Res_2.Service_Data_Response.Meas_Values_32Bit[PE_ID_COS_L2_MIN].Meas_Value;
                           #Driver_Data.Cos_L3_min := #V_PN_Meas_Data_Res_2.Service_Data_Response.Meas_Values_32Bit[PE_ID_COS_L3_MIN].Meas_Value;
                           #Driver_Data.Cos_Total_max := #V_PN_Meas_Data_Res_2.Service_Data_Response.Meas_Values_32Bit[PE_ID_COS_OVERALL_MAX].Meas_Value;
                           #Driver_Data.Cos_Total_min := #V_PN_Meas_Data_Res_2.Service_Data_Response.Meas_Values_32Bit[PE_ID_COS_OVERALL_MIN].Meas_Value;
                           #Driver_Data.S_L1_min := #V_PN_Meas_Data_Res_2.Service_Data_Response.Meas_Values_32Bit[PE_ID_S_L1_MIN].Meas_Value;
                           #Driver_Data.S_L2_min := #V_PN_Meas_Data_Res_2.Service_Data_Response.Meas_Values_32Bit[PE_ID_S_L2_MIN].Meas_Value;
                           #Driver_Data.S_L3_min := #V_PN_Meas_Data_Res_2.Service_Data_Response.Meas_Values_32Bit[PE_ID_S_L3_MIN].Meas_Value;
                           #Driver_Data.S_Total_max := #V_PN_Meas_Data_Res_2.Service_Data_Response.Meas_Values_32Bit[PE_ID_S_OVERALL_MAX].Meas_Value;
                           #Driver_Data.S_Total_min := #V_PN_Meas_Data_Res_2.Service_Data_Response.Meas_Values_32Bit[PE_ID_S_OVERALL_MIN].Meas_Value;
                           #Driver_Data.Q_L1_min := #V_PN_Meas_Data_Res_2.Service_Data_Response.Meas_Values_32Bit[PE_ID_Q_L1_MIN].Meas_Value;
                           #Driver_Data.Q_L2_min := #V_PN_Meas_Data_Res_2.Service_Data_Response.Meas_Values_32Bit[PE_ID_Q_L2_MIN].Meas_Value;
                           #Driver_Data.Q_L3_min := #V_PN_Meas_Data_Res_2.Service_Data_Response.Meas_Values_32Bit[PE_ID_Q_L3_MIN].Meas_Value;
                           #Driver_Data.Q_Total_max := #V_PN_Meas_Data_Res_2.Service_Data_Response.Meas_Values_32Bit[PE_ID_Q_OVERALL_MAX].Meas_Value;
                           #Driver_Data.Q_Total_min := #V_PN_Meas_Data_Res_2.Service_Data_Response.Meas_Values_32Bit[PE_ID_Q_OVERALL_MIN].Meas_Value;
                           #Driver_Data.P_L1_min := #V_PN_Meas_Data_Res_2.Service_Data_Response.Meas_Values_32Bit[PE_ID_P_L1_MIN].Meas_Value;
                           #Driver_Data.P_L2_min := #V_PN_Meas_Data_Res_2.Service_Data_Response.Meas_Values_32Bit[PE_ID_P_L2_MIN].Meas_Value;
                           #Driver_Data.P_L3_min := #V_PN_Meas_Data_Res_2.Service_Data_Response.Meas_Values_32Bit[PE_ID_P_L3_MIN].Meas_Value;
                           #Driver_Data.P_Total_max := #V_PN_Meas_Data_Res_2.Service_Data_Response.Meas_Values_32Bit[PE_ID_P_OVERALL_MAX].Meas_Value;
                           #Driver_Data.P_Total_min := #V_PN_Meas_Data_Res_2.Service_Data_Response.Meas_Values_32Bit[PE_ID_P_OVERALL_MIN].Meas_Value;
                       END_IF;

                       // Go to the state for waiting for the answer
                       #Sm_State_Next := #SM_IDLE;
                   ELSE
                       ; // Not ready yet
                   END_IF;

                   // Wait for the answer of the SENTRON PAC
               #SM_WRITE_MINMAX_WAIT_RESP:

                   // Start the watchdog, while waiting for a response
                   #Watchdog_Run := TRUE;

                   // The configuration of the data record 47 on the PAC 4200 failed with an error
                   IF ((#Write_Data_Record.ERROR = TRUE)
                       OR (#Watchdog.Q = TRUE)) THEN

                       // Reset the watchdog
                       #Watchdog_Run := FALSE;

                       // Save the error code for the user to display the error reason and location
                       #Error_Location := #ERR_LOC_WRITE_MIN_MAX_VALUES;
                       #Error_Code := #Write_Data_Record.STATUS;

                       // Reset the request bit to write a record to the Energy Meter for
                       // generating a positive edge with the next request
                       #Write_Data_Rec_Request := FALSE;

                       // Release the communication resource
                       #Comm_Resource_Counter := #Comm_Resource_Counter - 1;

                       // Go back to the main state and wait for a new request
                       #Sm_State_Next := #SM_IDLE;

                       // The configuration of the data record 47 on the PAC 4200 has been finished with success
                   ELSIF (#Write_Data_Record.DONE = TRUE) THEN

                       // Reset the watchdog
                       #Watchdog_Run := FALSE;

                       // Reset the error code and location
                       #Error_Code := DW#16#0000_0000;

                       // Reset the request bit to write a record to the SENTRON PAC 4200 for
                       // generating a positive edge with the next request
                       #Write_Data_Rec_Request := FALSE;

                       // Now configure the values to read these measurement values
                       #Rd_Rec_Index := 47;
                       #Rd_Rec_Max_Length := 232;

                       // Start the reading of the measurement values
                       #Read_Data_Rec_Request := TRUE;

                       // Go back to the main state and wait for a new request
                       #Sm_State_Next := #SM_READ_MINMAX_WAIT_RESP;
                   ELSE
                       ; // Reading still in progress
                   END_IF;

                   // Wait for an answer of the reading of the min max values
               #SM_READ_MINMAX_WAIT_RESP:

                   // Start the watchdog, while waiting for a response
                   #Watchdog_Run := TRUE;

                   // Set the request to true, if the bit is reset in case of an error
                   #Read_Data_Rec_Request := #Error_Retry_Timer.Q;

                   // The update of the data failed with an error
                   IF ((#Read_Data_Record.ERROR = TRUE)
                       OR (#Watchdog.Q = TRUE)) THEN

                       // Reset the request bit to read a record from the Energy Meter for
                       // generating a positive edge with the next request
                       #Read_Data_Rec_Request := FALSE;

                       // Increase the retries to get an answer
                       #Error_Retry_Counter := #Error_Retry_Counter + 1;

                       // Check if the device is still busy
                       IF (((#Read_Data_Record.STATUS = #ERROR_CODE_DEVICE_BUSY)
                           AND (#Error_Retry_Counter >= #ERROR_RETRY_LIMIT))
                           OR (#Read_Data_Record.STATUS <> #ERROR_CODE_DEVICE_BUSY)) THEN

                           // Reset the watchdog
                           #Watchdog_Run := FALSE;

                           // Save the time to update the values, even with an error
                           #Time_to_update := #Time_Measurement.ET;

                           // Reset the timer to restart the time next time
                           #Time_Measurement(IN := FALSE,
                                             PT := T#21d);

                           // Reset the timer
                           #Error_Retry_Timer_Run := FALSE;

                           // Reset the retry counter
                           #Error_Retry_Counter := 0;

                           // Save the error code for the user to display the error reason and location
                           #Error_Location := #ERR_LOC_READ_MIN_MAX_VALUES;
                           #Error_Code := #Read_Data_Record.STATUS;

                           // Release the communication resource
                           #Comm_Resource_Counter := #Comm_Resource_Counter - 1;

                           // Go back to the main state and wait for a new request
                           #Sm_State_Next := #SM_IDLE;
                       ELSE
                           // Reset the timer
                           #Error_Retry_Timer(IN := FALSE,
                                              PT := #TIME_RETRY_TIMER);

                           // Start the error timer
                           #Error_Retry_Timer_Run := TRUE;
                       END_IF;

                       // The update of the has been finished with success
                   ELSIF (#Read_Data_Record.VALID = TRUE) THEN

                       // Reset the watchdog
                       #Watchdog_Run := FALSE;

                       // Reset the retry counter
                       #Error_Retry_Counter := 0;

                       // Reset the error code and location
                       #Error_Code := DW#16#0000_0000;

                       // Save the time to update the values
                       #Time_to_update := #Time_Measurement.ET;

                       // Reset the timer to restart the time next time
                       #Time_Measurement(IN := FALSE,
                                         PT := T#21d);

                       // Read the current time to set the timestamp of the measurement values
                       #General_Ret_Val := RD_SYS_T(OUT => #Time_Stamp_Meas_Values);

                       // Release the communication resource
                       #Comm_Resource_Counter := #Comm_Resource_Counter - 1;

                       // Reset the request bit to read a record from the Energy Meter for
                       // generating a positive edge with the next request
                       #Read_Data_Rec_Request := FALSE;

                       // The default value for a not measured value is DW16FFFF_FFFF
                       // ==> replace it with 0.0
                       // ==> Therefore check every value in a FOR-loop if it is the default value
                       FOR #Index := 1 TO 58 BY 1 DO
                           IF (#V_DP_Min_Max_Reset.Meas_Values[#Index] = DW#16#FFFF_FFFF) THEN
                               #V_DP_Min_Max_Reset.Meas_Values[#Index] := DW#16#0;
                           ELSE
                               ; // Value is correct
                           END_IF;
                       END_FOR;

                       //===========================================================================
                       //====== Generate the minimum and maximum values ============================
                       //===========================================================================

                       // ================================================
                       // Proceed the voltage values for each phase
                       // ================================================
                       #Driver_Data.U_L1_max := #V_DP_Meas_Min_Max.U_L1_Max;
                       #Driver_Data.U_L1_min := #V_DP_Meas_Min_Max.U_L1_Min;
                       #Driver_Data.U_L2_max := #V_DP_Meas_Min_Max.U_L2_Max;
                       #Driver_Data.U_L2_min := #V_DP_Meas_Min_Max.U_L2_Min;
                       #Driver_Data.U_L3_max := #V_DP_Meas_Min_Max.U_L3_Max;
                       #Driver_Data.U_L3_min := #V_DP_Meas_Min_Max.U_L3_Min;
                       #Driver_Data.U_PH_N_Average_max := #V_DP_Meas_Min_Max.U_PH_N_Average_Max;
                       #Driver_Data.U_PH_N_Average_min := #V_DP_Meas_Min_Max.U_PH_N_Average_Min;

                       // ================================================
                       // Proceed the voltage values for phase to phase
                       // ================================================
                       #Driver_Data.U_L1_L2_max := #V_DP_Meas_Min_Max.U_L1_L2_Max;
                       #Driver_Data.U_L1_L2_min := #V_DP_Meas_Min_Max.U_L1_L2_Min;
                       #Driver_Data.U_L2_L3_max := #V_DP_Meas_Min_Max.U_L2_L3_Max;
                       #Driver_Data.U_L2_L3_min := #V_DP_Meas_Min_Max.U_L2_L3_Min;
                       #Driver_Data.U_L3_L1_max := #V_DP_Meas_Min_Max.U_L3_L1_Max;
                       #Driver_Data.U_L3_L1_min := #V_DP_Meas_Min_Max.U_L3_L1_Min;
                       #Driver_Data.U_PH_PH_Average_max := #V_DP_Meas_Min_Max.U_PH_PH_Average_Max;
                       #Driver_Data.U_PH_PH_Average_min := #V_DP_Meas_Min_Max.U_PH_PH_Average_Min;

                       // ================================================
                       // Proceed the current for each phase
                       // ================================================
                       #Driver_Data.I_L1_max := #V_DP_Meas_Min_Max.I_L1_Max;
                       #Driver_Data.I_L1_min := #V_DP_Meas_Min_Max.I_L1_Min;
                       #Driver_Data.I_L2_max := #V_DP_Meas_Min_Max.I_L2_Max;
                       #Driver_Data.I_L2_min := #V_DP_Meas_Min_Max.I_L2_Min;
                       #Driver_Data.I_L3_max := #V_DP_Meas_Min_Max.I_L3_Max;
                       #Driver_Data.I_L3_min := #V_DP_Meas_Min_Max.I_L3_Min;
                       #Driver_Data.I_Average_max := #V_DP_Meas_Min_Max.I_Average_Max;
                       #Driver_Data.I_Average_min := #V_DP_Meas_Min_Max.I_Average_Min;

                       // ================================================
                       // Proceed the frequency for the complete net
                       // ================================================
                       #Driver_Data.f_max := #V_DP_Meas_Min_Max.f_Max;
                       #Driver_Data.f_min := #V_DP_Meas_Min_Max.f_Min;

                       // ================================================
                       // Proceed the cos for each phase
                       // ================================================
                       #Driver_Data.Cos_L1_max := #V_DP_Meas_Min_Max.Cos_L1_Max;
                       #Driver_Data.Cos_L1_min := #V_DP_Meas_Min_Max.Cos_L1_Min;
                       #Driver_Data.Cos_L2_max := #V_DP_Meas_Min_Max.Cos_L2_Max;
                       #Driver_Data.Cos_L2_min := #V_DP_Meas_Min_Max.Cos_L2_Min;
                       #Driver_Data.Cos_L3_max := #V_DP_Meas_Min_Max.Cos_L3_Max;
                       #Driver_Data.Cos_L3_min := #V_DP_Meas_Min_Max.Cos_L3_Min;
                       #Driver_Data.Cos_Total_max := #V_DP_Meas_Min_Max.Cos_Total_Max;
                       #Driver_Data.Cos_Total_min := #V_DP_Meas_Min_Max.Cos_Total_Min;

                       // ================================================
                       // Proceed the apparent power for each phase
                       // ================================================
                       #Driver_Data.S_L1_max := #V_DP_Meas_Min_Max.S_L1_Max;
                       #Driver_Data.S_L1_min := #V_DP_Meas_Min_Max.S_L1_Min;
                       #Driver_Data.S_L2_max := #V_DP_Meas_Min_Max.S_L2_Max;
                       #Driver_Data.S_L2_min := #V_DP_Meas_Min_Max.S_L2_Min;
                       #Driver_Data.S_L3_max := #V_DP_Meas_Min_Max.S_L3_Max;
                       #Driver_Data.S_L3_min := #V_DP_Meas_Min_Max.S_L3_Min;
                       #Driver_Data.S_Total_max := #V_DP_Meas_Min_Max.S_Total_Max;
                       #Driver_Data.S_Total_min := #V_DP_Meas_Min_Max.S_Total_Min;

                       // ================================================
                       // Proceed the reactive power for each phase
                       // ================================================
                       #Driver_Data.Q_L1_max := #V_DP_Meas_Min_Max.Q_L1_Max;
                       #Driver_Data.Q_L1_min := #V_DP_Meas_Min_Max.Q_L1_Min;
                       #Driver_Data.Q_L2_max := #V_DP_Meas_Min_Max.Q_L2_Max;
                       #Driver_Data.Q_L2_min := #V_DP_Meas_Min_Max.Q_L2_Min;
                       #Driver_Data.Q_L3_max := #V_DP_Meas_Min_Max.Q_L3_Max;
                       #Driver_Data.Q_L3_min := #V_DP_Meas_Min_Max.Q_L3_Min;
                       #Driver_Data.Q_Total_max := #V_DP_Meas_Min_Max.Q_Total_Max;
                       #Driver_Data.Q_Total_min := #V_DP_Meas_Min_Max.Q_Total_Min;

                       // ================================================
                       // Proceed the effective power for each phase
                       // ================================================
                       #Driver_Data.P_L1_max := #V_DP_Meas_Min_Max.P_L1_Max;
                       #Driver_Data.P_L1_min := #V_DP_Meas_Min_Max.P_L1_Min;
                       #Driver_Data.P_L2_max := #V_DP_Meas_Min_Max.P_L2_Max;
                       #Driver_Data.P_L2_min := #V_DP_Meas_Min_Max.P_L2_Min;
                       #Driver_Data.P_L3_max := #V_DP_Meas_Min_Max.P_L3_Max;
                       #Driver_Data.P_L3_min := #V_DP_Meas_Min_Max.P_L3_Min;
                       #Driver_Data.P_Total_max := #V_DP_Meas_Min_Max.P_Total_Max;
                       #Driver_Data.P_Total_min := #V_DP_Meas_Min_Max.P_Total_Min;

                       // Go back to the main state and wait for a new request
                       #Sm_State_Next := #SM_IDLE;
                   ELSE
                       ; // Reading still in progress
                   END_IF;
           END_CASE;

           // Set information for the visualization block
           #Driver_Data.Read_Value := #Automatic_Update;
           #Driver_Data.Driver_Error := BOOL_TO_INT(#Error_Code <> 0);
           #Driver_Data.Connection_Type := #Connection_Type;

           // Store the value for edge detection
           #Start_Acyclic_HMI_Old := #HMI_Bits_Internal.Start_Acyclic;
           #Reset_Energy_Old := #Reset_Energy_Counter;
           #Reset_Energy_HMI_Old := #HMI_Bits_Internal.Reset_Energy_Meter;
           #Reset_Min_Max_Old := #Reset_Min_Max;
           #Reset_Min_Max_HMI_Old := #HMI_Bits_Internal.Reset_min_max_Data;

       END_IF;
END_FUNCTION_BLOCK
